PROGRAM PRG_FiberLite
VAR
END_VAR

// Set LED output scaling (Fiber-Lite)
bLedOutput1.iTermBits := 14;
bLedOutput1(fbSetIllPercent=>);

END_PROGRAM

(* stored: Version 1.1.0.1, ProductVersion 3.1.4022.18
   POU PRG_FiberLite: Id {f77f6f57-8f90-4848-b1bb-153be6bbff26}, SpecialFunc None *)
